INTERFACE I_LimitedStringBuilder

METHOD Append : I_StringBuilder
VAR_INPUT
	sText	: T_MaxString;
END_VAR
END_METHOD

METHOD Reset : I_LimitedStringBuilder
VAR_INPUT
END_VAR
END_METHOD

METHOD ToString : T_MaxString
VAR_INPUT
END_VAR
END_METHOD

END_INTERFACE

(* stored: Version 1.1.0.1
   Itf I_LimitedStringBuilder: Id {fcf763eb-9252-4017-a88f-d8e76fd5cb3c}
   Method Append: Id {02be178d-9282-45e4-9d7f-cae966472eb0}
   Method Reset: Id {3551b35a-fbb0-4435-804f-a402d1cc4ae0}
   Method ToString: Id {5460b69e-09ae-43b2-9de8-f996467d7fc0} *)
